{attribute 'GeneratedUsingTerminal: EL1258-0000-0016'}
{attribute addProperty BoxType "EL1258-0000-0016"}
{attribute addProperty Id "StatusAT %I*Status_56B69FDC6InputsAT %I*Inputs_62625F9410Input_event_timeAT %I*ARRAY[0..9] OF UDINT40"}
{attribute addProperty CRC "827289277"}
{attribute addProperty Size "56"}
TYPE MTI_Inputs_10x_Channel_C3ED30FD :
STRUCT
	{attribute addProperty Name "Status"}
	Status AT %I* : Status_56B69FDC;
	{attribute addProperty Name "Inputs"}
	Inputs AT %I* : Inputs_62625F94;
	{attribute addProperty Name "Input_event_time"}
	Input_event_time AT %I* : ARRAY[0..9] OF UDINT;
END_STRUCT
END_TYPE

(* stored: Version 1.2.0.0, ProductVersion 3.1.4024.9
   DUT MTI_Inputs_10x_Channel_C3ED30FD: Id {239bb938-557b-443e-982b-7807c5deedc6} *)
